FUNCTION_BLOCK FB_ENCODER_V3
VAR_OUTPUT
	THETA_EL 			: REAL;
	THETA_MECH 			: REAL;
	OMEGA_EL 			: REAL;
	OMEGA_MECH 			: REAL;
END_VAR
VAR
	COUNTER_MAX 		: UINT := 16383;
	COUNTER_INV_MAX 	: UINT := 65535;
	COUNTER_TEMP 		: UINT;
	SAMPLE_TIME			: REAL := 100E-6;
END_VAR
VAR_STAT
   	THETA_MECH_PREV 	: REAL := 0;
END_VAR


// If counter is maximum UINT value (or over COUNTER_MAX), rotation is reversed.
IF Measurements.COUNTER_VALUE > COUNTER_MAX THEN
	COUNTER_TEMP := COUNTER_MAX + (Measurements.COUNTER_VALUE - COUNTER_INV_MAX);
ELSE
	COUNTER_TEMP := Measurements.COUNTER_VALUE;
END_IF

IF Measurements.COUNTER_VALUE >= Measurements.COUNTER_OFFSET THEN
	COUNTER_TEMP := COUNTER_TEMP - Measurements.COUNTER_OFFSET;
ELSIF Measurements.COUNTER_VALUE < Measurements.COUNTER_OFFSET THEN
	COUNTER_TEMP := COUNTER_TEMP + Measurements.COUNTER_OFFSET;
END_IF

IF COUNTER_TEMP > COUNTER_MAX THEN
	COUNTER_TEMP := COUNTER_MAX;
END_IF

THETA_MECH := LREAL_TO_REAL(2*PI*UINT_TO_LREAL(COUNTER_TEMP)/UINT_TO_LREAL(COUNTER_MAX));

IF THETA_MECH*2 > 2*PI THEN
	THETA_EL := LREAL_TO_REAL(THETA_MECH*2 - 2*PI);
ELSE
	THETA_EL := THETA_MECH*2;
END_IF

OMEGA_MECH := (THETA_MECH-THETA_MECH_PREV)/SAMPLE_TIME;
THETA_MECH_PREV := THETA_MECH;

OMEGA_EL := OMEGA_MECH*2;

END_FUNCTION_BLOCK

(* stored: Version 1.1.0.1, ProductVersion 3.1.4024.11
   POU FB_ENCODER_V3: Id {d4ab4016-1b5f-4278-a9df-608ca632a5aa}, SpecialFunc None *)
